PROGRAM main
VAR_INPUT
	X0 : bool;
	X1 : bool;
	X2 : bool;
END_VAR

VAR_OUTPUT
	Y0 : bool;
END_VAR

VAR
	M0 : bool;
	M1 : bool;
END_VAR

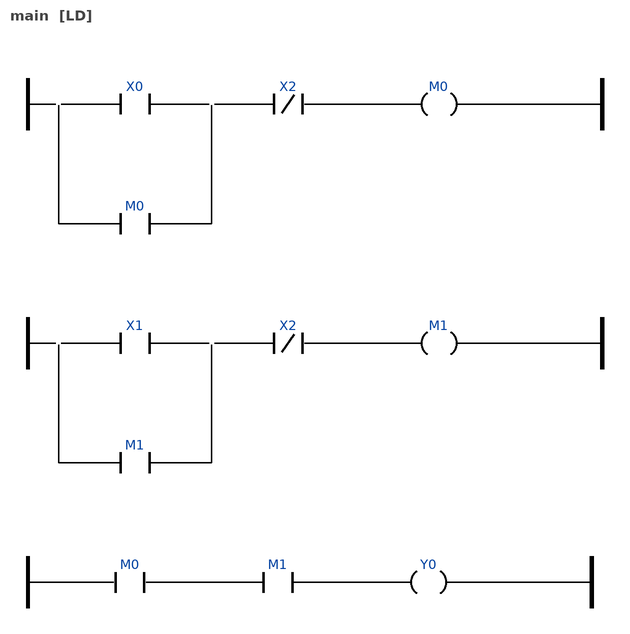
(* LD diagram, written out as Structured Text *)
M0 := (X0 OR M0) AND NOT X2;
M1 := (X1 OR M1) AND NOT X2;
Y0 := M0 AND M1;
END_PROGRAM
